// TIA Portal V18 export
FUNCTION_BLOCK "_spot_iteratorWaitForXray"   // FB33, FBD
{ S7_Optimized_Access := 'TRUE' }
VERSION : 0.1
// stored: AutoNumber true, IsIECCheckEnabled false, IsRetainMemResEnabled false, MemoryReserve 100, SetENOAutomatically false, UDAEnableTagReadback false
   VAR_INPUT
      ALLOWED : Bool;
      xButtonStartAuto : Bool;
      motors_all_arrived : Bool;
      XRAY_SHOT_DONE : Bool;
      Spot_i_maxN : Int;
      sec_siren_done : Real := 2.0;
   END_VAR
   VAR_OUTPUT
      reset_PC_SHOT_DONE : Bool;
      state_comment : WString;
      cycleActive : Bool;
      motos_go_now_command : Bool;
      XRAY_READYFORSHOT : Bool;
      ySirenDone : Bool;
   END_VAR
   VAR_IN_OUT
      spot_i : Int;
      state : UInt;
   END_VAR
   VAR
      pt_siren_done { ExternalAccessible := 'False'; ExternalVisible := 'False'; ExternalWritable := 'False'} : Time := T#1s;
      mem1 : Bool;
      mem2 : Bool;
      tons12 { S7_SetPoint := 'True'} : TON_TIME;
      tons20 { S7_SetPoint := 'True'} : TON_TIME;
      tons10 { S7_SetPoint := 'True'} : TON_TIME;
      pt_xray_stuck_in_done { ExternalAccessible := 'False'; ExternalVisible := 'False'; ExternalWritable := 'False'} : Time := T#1s;
      pt_mot_delay : Time := T#100ms;
      tons20a { S7_SetPoint := 'True'} : TON_TIME;
      tons24 { S7_SetPoint := 'True'} : TON_TIME;
      mem3 : Bool;
   END_VAR
   VAR_TEMP
      temp_be_going_to_next_SPOT : Bool;
      temp_be_going_home : Bool;
      reset_pc_shot_done_s20 : Bool;
      reset_pc_shot_done_s23 : Bool;
      queEndReached : Bool;
   END_VAR
   VAR CONSTANT
      s0wait : UInt := 0;
      s20NextPositionGoCommand : UInt := 20;
      s21NextPositionGoing : UInt := 21;
      s22NextPositionArrivedWaitingForXrayPicture : UInt := 22;
      s23NextPositionIncrement : UInt := 23;
      s24NextPositionDone : UInt := 24;
      wstrings00wait : WString := WSTRING#'Ожидание';
      wstrings20NextPositionGoCommand_1 : WString := WSTRING#'Движение к следующей позиции';
      wstrings21NextPositionGoing_1 : WString := WSTRING#'Движение к следующей позиции';
      wstrings22NextPositionArrivedWaitingForXrayPicture_1 : WString := WSTRING#'ожидание снимка';
      wstrings23NextPositionIncrement_1 : WString := WSTRING#'увеличение индекса позиции';
      wstrings24NextPositionDone_1 : WString := WSTRING#'Цикл завершен';
      CELL_INDEX_HOME : UInt := 1;
      Spot_index_start : UInt := 1;
   END_VAR
   VAR_TEMP   // added for the SCL form of the ladder/FBD networks
      _w1 : Bool;
      _w2 : Bool;
      _w3 : Bool;
      _w4 : Bool;
   END_VAR
BEGIN

REGION Network 3
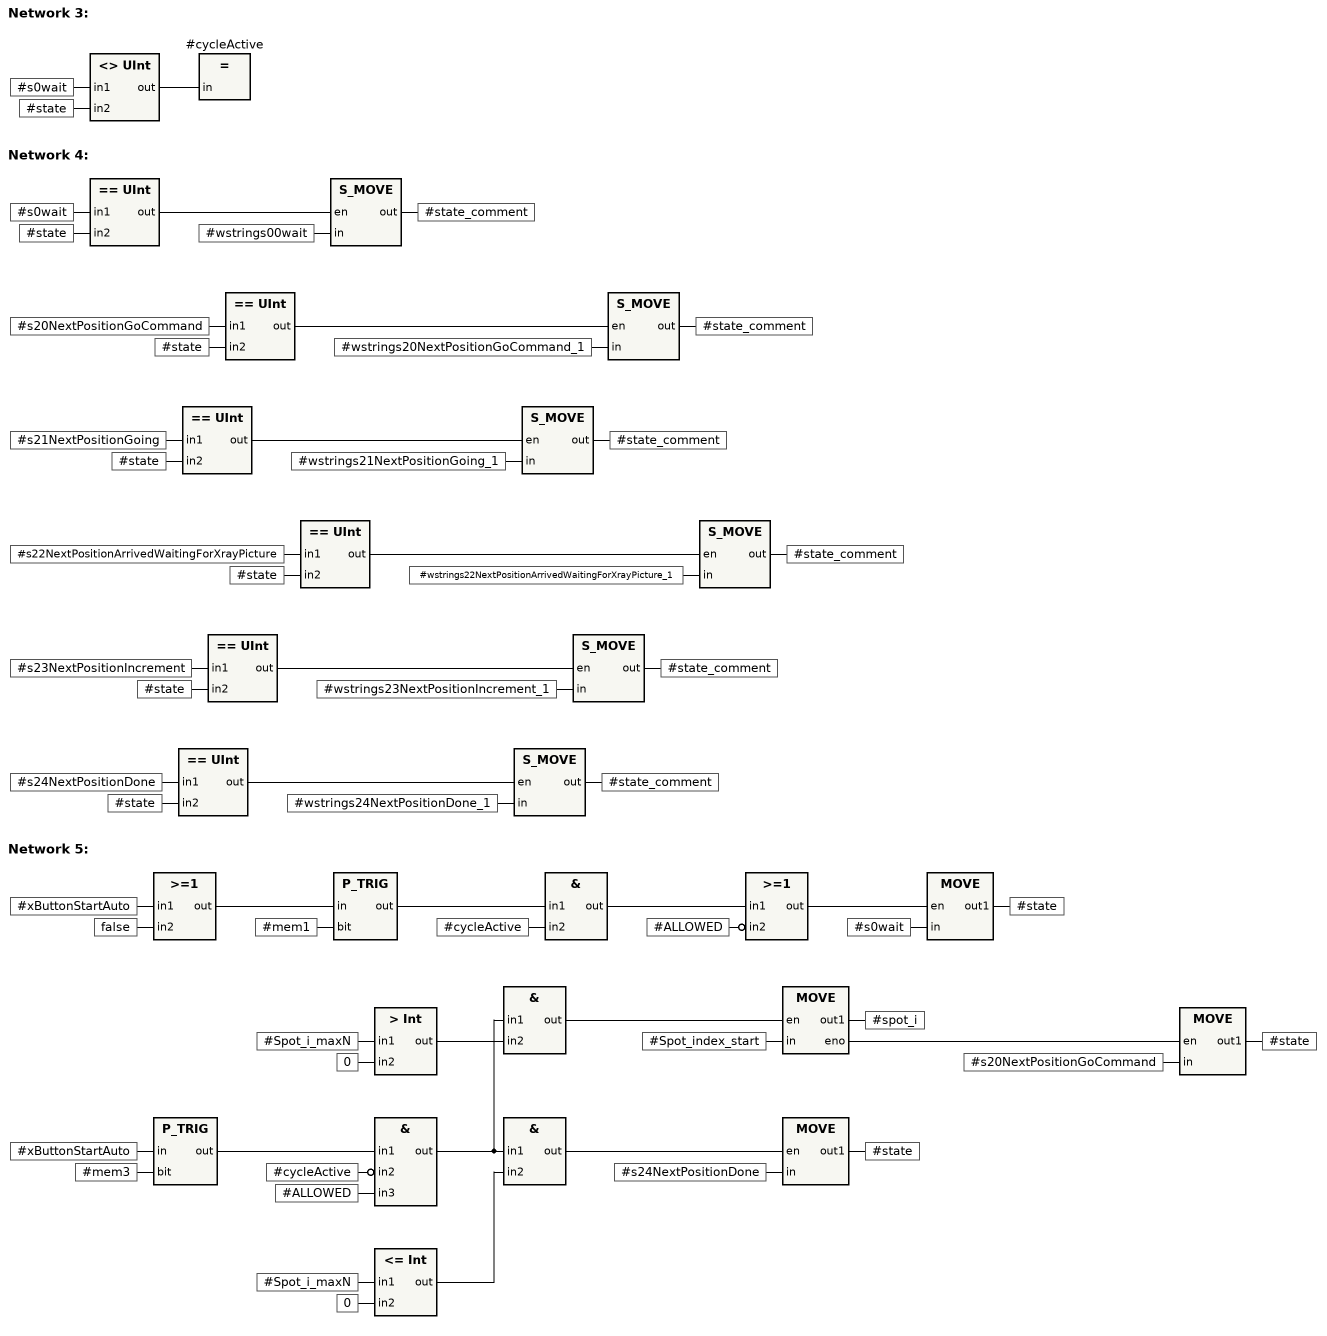
   #cycleActive := #s0wait <> #state;
END_REGION

REGION Network 4
   IF #s0wait = #state THEN #state_comment := #wstrings00wait; END_IF;
   IF #s20NextPositionGoCommand = #state THEN #state_comment := #wstrings20NextPositionGoCommand_1; END_IF;
   IF #s21NextPositionGoing = #state THEN #state_comment := #wstrings21NextPositionGoing_1; END_IF;
   IF #s22NextPositionArrivedWaitingForXrayPicture = #state THEN
       #state_comment := #wstrings22NextPositionArrivedWaitingForXrayPicture_1;
   END_IF;
   IF #s23NextPositionIncrement = #state THEN #state_comment := #wstrings23NextPositionIncrement_1; END_IF;
   IF #s24NextPositionDone = #state THEN #state_comment := #wstrings24NextPositionDone_1; END_IF;
END_REGION

REGION Network 5
   #_w1 := #xButtonStartAuto OR false;
   #_w2 := #_w1 AND NOT #mem1;   // rising edge
   #mem1 := #_w1;
   IF (#_w2 AND #cycleActive) OR NOT #ALLOWED THEN #state := #s0wait; END_IF;
   #_w3 := #xButtonStartAuto AND NOT #mem3;   // rising edge
   #mem3 := #xButtonStartAuto;
   #_w4 := #_w3 AND NOT #cycleActive AND #ALLOWED;
   IF #_w4 AND (#Spot_i_maxN > 0) THEN
       #spot_i := #Spot_index_start;
       #state := #s20NextPositionGoCommand;
   END_IF;
   IF #_w4 AND (#Spot_i_maxN <= 0) THEN #state := #s24NextPositionDone; END_IF;
END_REGION

REGION Network 6
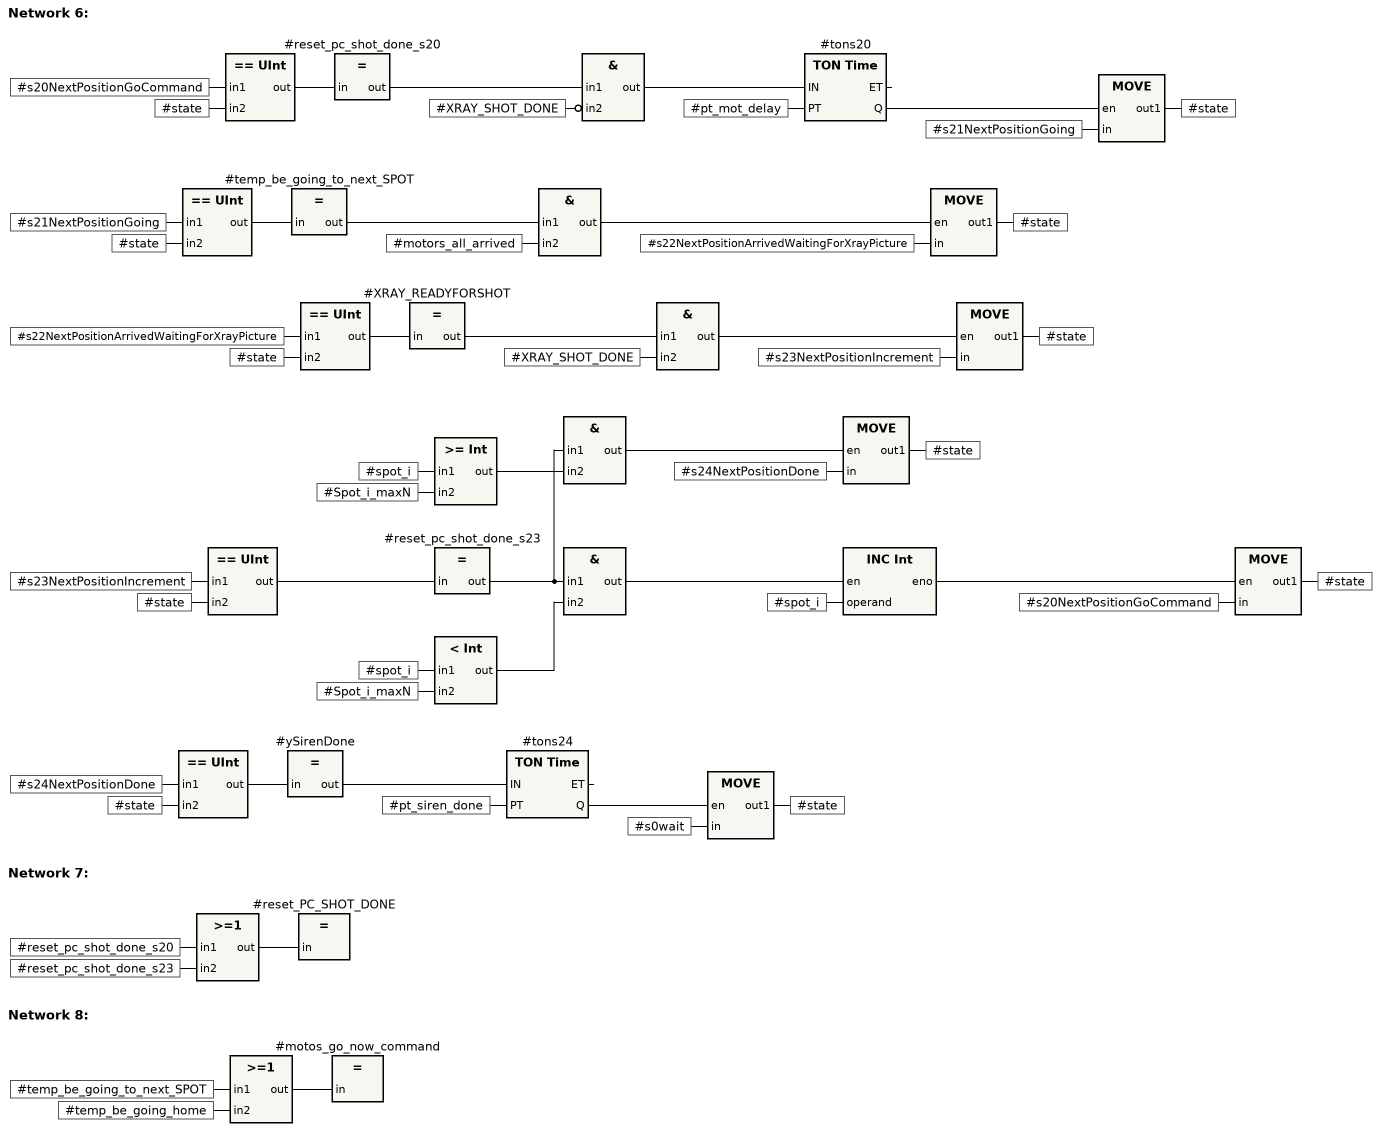
   #reset_pc_shot_done_s20 := #s20NextPositionGoCommand = #state;
   #tons20(IN := #reset_pc_shot_done_s20 AND NOT #XRAY_SHOT_DONE, PT := #pt_mot_delay);   // TON
   IF #tons20.Q THEN #state := #s21NextPositionGoing; END_IF;
   #temp_be_going_to_next_SPOT := #s21NextPositionGoing = #state;
   IF #temp_be_going_to_next_SPOT AND #motors_all_arrived THEN
       #state := #s22NextPositionArrivedWaitingForXrayPicture;
   END_IF;
   #XRAY_READYFORSHOT := #s22NextPositionArrivedWaitingForXrayPicture = #state;
   IF #XRAY_READYFORSHOT AND #XRAY_SHOT_DONE THEN #state := #s23NextPositionIncrement; END_IF;
   #reset_pc_shot_done_s23 := #s23NextPositionIncrement = #state;
   IF #reset_pc_shot_done_s23 AND (#spot_i >= #Spot_i_maxN) THEN #state := #s24NextPositionDone; END_IF;
   #_w1 := #reset_pc_shot_done_s23 AND (#spot_i < #Spot_i_maxN);
   IF #_w1 THEN
       #spot_i := #spot_i + 1;
       #state := #s20NextPositionGoCommand;
   END_IF;
   #ySirenDone := #s24NextPositionDone = #state;
   #tons24(IN := #ySirenDone, PT := #pt_siren_done);   // TON
   IF #tons24.Q THEN #state := #s0wait; END_IF;
END_REGION

REGION Network 7
   #reset_PC_SHOT_DONE := #reset_pc_shot_done_s20 OR #reset_pc_shot_done_s23;
END_REGION

REGION Network 8
   #motos_go_now_command := #temp_be_going_to_next_SPOT OR #temp_be_going_home;
END_REGION

REGION Network 9 (SCL)
   #pt_siren_done := REAL_TO_DINT(#sec_siren_done * 1000);
END_REGION
END_FUNCTION_BLOCK
